% RSLogix 500 project P4_BAK000.RSS, saved by version 8.10.00.18 %
PROJECT "UNTITLED"    % processor: MicroLogix 1200 %

PROGRAM FILES
  LAD 2   4 rungs
  LAD 3 "IO'S"  7 rungs
  LAD 4 "CONTROL"  11 rungs
  LAD 5 "CYCLE'S"  10 rungs

DATA FILES
  O0 OUTPUT  4 elements
  I1 INPUT  4 elements
  S2 STATUS  66 elements
  B3 BINARY  2 elements
  T4 TIMER  3 elements
  C5 COUNTER  1 elements
  R6 CONTROL  1 elements
  N7 INTEGER  2 elements

LADDER 2
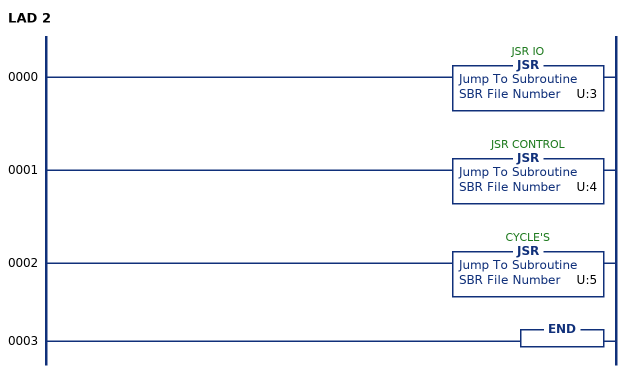
% Rung: 0 %
SOR JSR U:3 EOR
%   U:3  "JSR IO" %
% Rung: 1 %
SOR JSR U:4 EOR
%   U:4  "JSR CONTROL" %
% Rung: 2 %
SOR JSR U:5 EOR
%   U:5  "CYCLE'S" %
% Rung: 3 %
SOR END EOR

LADDER 3 "IO'S"
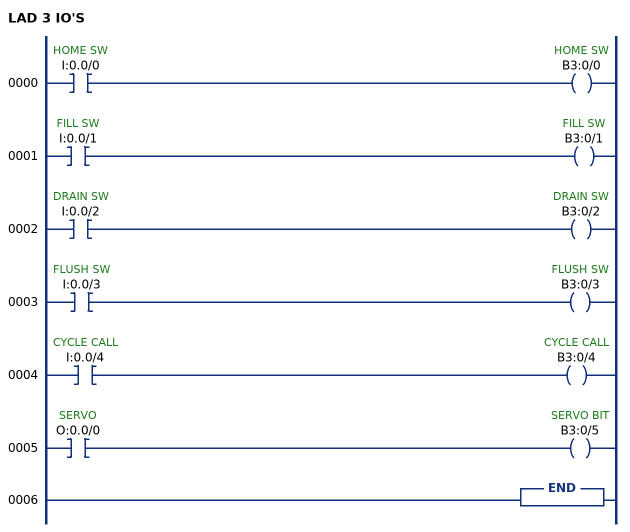
% Rung: 0 %
SOR XIC I:0.0/0 OTE B3:0/0 EOR
%   I:0.0/0  "HOME SW" %
%   B3:0/0  "HOME SW" %
% Rung: 1 %
SOR XIC I:0.0/1 OTE B3:0/1 EOR
%   I:0.0/1  "FILL SW" %
%   B3:0/1  "FILL SW" %
% Rung: 2 %
SOR XIC I:0.0/2 OTE B3:0/2 EOR
%   I:0.0/2  "DRAIN SW" %
%   B3:0/2  "DRAIN SW" %
% Rung: 3 %
SOR XIC I:0.0/3 OTE B3:0/3 EOR
%   I:0.0/3  "FLUSH SW" %
%   B3:0/3  "FLUSH SW" %
% Rung: 4 %
SOR XIC I:0.0/4 OTE B3:0/4 EOR
%   I:0.0/4  "CYCLE CALL" %
%   B3:0/4  "CYCLE CALL" %
% Rung: 5 %
SOR XIC O:0.0/0 OTE B3:0/5 EOR
%   O:0.0/0  "SERVO" %
%   B3:0/5  "SERVO BIT" %
% Rung: 6 %
SOR END EOR

LADDER 4 "CONTROL"
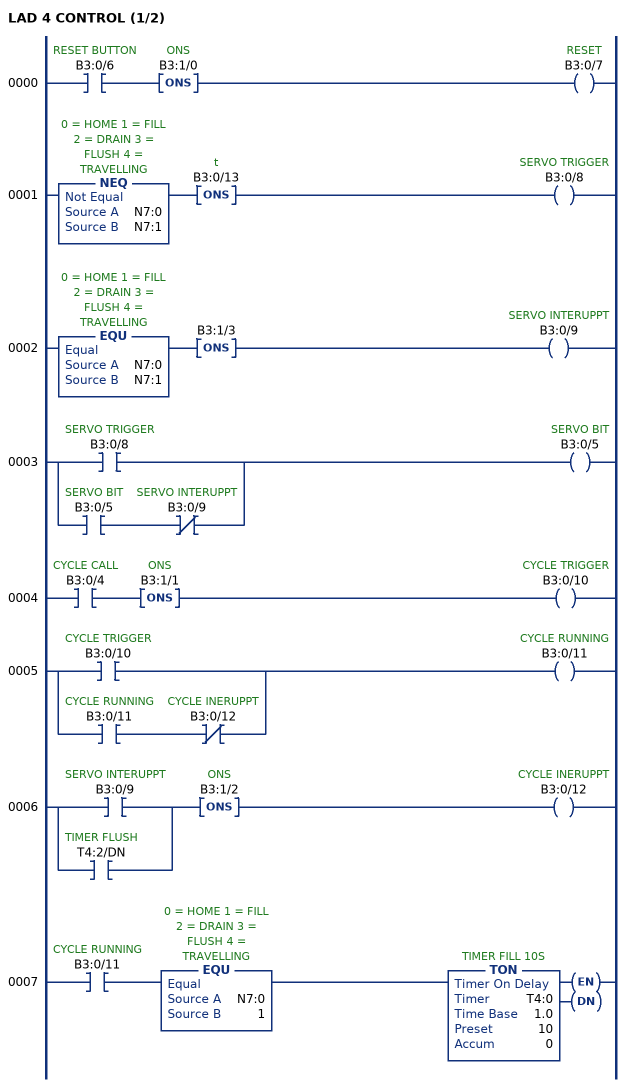
% Rung: 0 %
SOR XIC B3:0/6 ONS B3:1/0 OTE B3:0/7 EOR
%   B3:0/6  "RESET BUTTON" %
%   B3:1/0  "ONS" %
%   B3:0/7  "RESET" %
% Rung: 1 %
SOR NEQ N7:0 N7:1 ONS B3:0/13 OTE B3:0/8 EOR
%   N7:0  "0 = HOME 1 = FILL 2 = DRAIN 3 = FLUSH 4 = TRAVELLING" %
%   N7:1  "DESIRED:    0 = HOME 1 = FILL 2 = DRAIN 3 = FLUSH 4 = TRAVELLING" %
%   B3:0/13  "t" %
%   B3:0/8  "SERVO TRIGGER" %
% Rung: 2 %
SOR EQU N7:0 N7:1 ONS B3:1/3 OTE B3:0/9 EOR
%   N7:0  "0 = HOME 1 = FILL 2 = DRAIN 3 = FLUSH 4 = TRAVELLING" %
%   N7:1  "DESIRED:    0 = HOME 1 = FILL 2 = DRAIN 3 = FLUSH 4 = TRAVELLING" %
%   B3:0/9  "SERVO INTERUPPT" %
% Rung: 3 %
SOR BST XIC B3:0/8 NXB XIC B3:0/5 XIO B3:0/9 BND OTE B3:0/5 EOR
%   B3:0/8  "SERVO TRIGGER" %
%   B3:0/5  "SERVO BIT" %
%   B3:0/9  "SERVO INTERUPPT" %
% Rung: 4 %
SOR XIC B3:0/4 ONS B3:1/1 OTE B3:0/10 EOR
%   B3:0/4  "CYCLE CALL" %
%   B3:1/1  "ONS" %
%   B3:0/10  "CYCLE TRIGGER" %
% Rung: 5 %
SOR BST XIC B3:0/10 NXB XIC B3:0/11 XIO B3:0/12 BND OTE B3:0/11 EOR
%   B3:0/10  "CYCLE TRIGGER" %
%   B3:0/11  "CYCLE RUNNING" %
%   B3:0/12  "CYCLE INERUPPT" %
% Rung: 6 %
SOR BST XIC B3:0/9 NXB XIC T4:2/DN BND ONS B3:1/2 OTE B3:0/12 EOR
%   B3:0/9  "SERVO INTERUPPT" %
%   T4:2  "TIMER FLUSH" %
%   B3:1/2  "ONS" %
%   B3:0/12  "CYCLE INERUPPT" %
% Rung: 7 %
SOR XIC B3:0/11 EQU N7:0 1 TON T4:0 1.0 10 0 EOR
%   B3:0/11  "CYCLE RUNNING" %
%   N7:0  "0 = HOME 1 = FILL 2 = DRAIN 3 = FLUSH 4 = TRAVELLING" %
%   T4:0  "TIMER FILL 10S" %

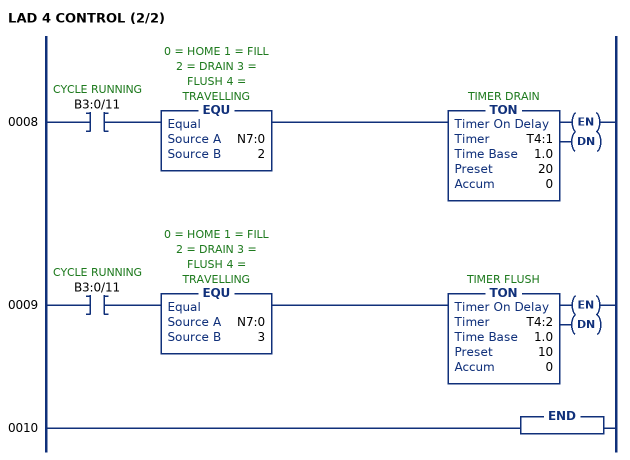
% Rung: 8 %
SOR XIC B3:0/11 EQU N7:0 2 TON T4:1 1.0 20 0 EOR
%   B3:0/11  "CYCLE RUNNING" %
%   N7:0  "0 = HOME 1 = FILL 2 = DRAIN 3 = FLUSH 4 = TRAVELLING" %
%   T4:1  "TIMER DRAIN" %
% Rung: 9 %
SOR XIC B3:0/11 EQU N7:0 3 TON T4:2 1.0 10 0 EOR
%   B3:0/11  "CYCLE RUNNING" %
%   N7:0  "0 = HOME 1 = FILL 2 = DRAIN 3 = FLUSH 4 = TRAVELLING" %
%   T4:2  "TIMER FLUSH" %
% Rung: 10 %
SOR END EOR

LADDER 5 "CYCLE'S"
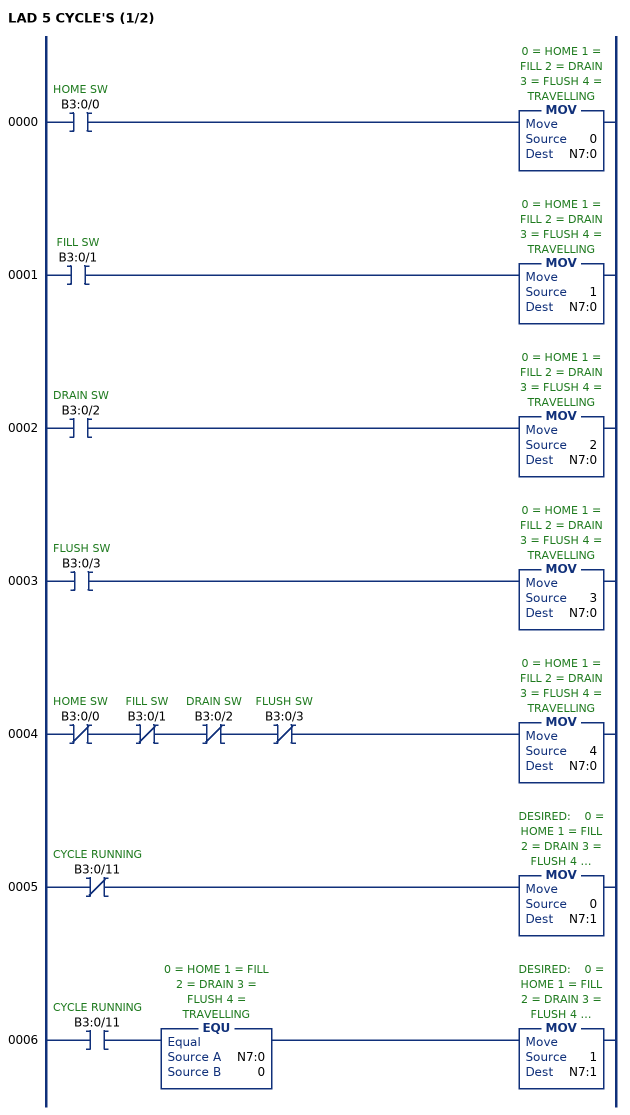
% Rung: 0 %
SOR XIC B3:0/0 MOV 0 N7:0 EOR
%   B3:0/0  "HOME SW" %
%   N7:0  "0 = HOME 1 = FILL 2 = DRAIN 3 = FLUSH 4 = TRAVELLING" %
% Rung: 1 %
SOR XIC B3:0/1 MOV 1 N7:0 EOR
%   B3:0/1  "FILL SW" %
%   N7:0  "0 = HOME 1 = FILL 2 = DRAIN 3 = FLUSH 4 = TRAVELLING" %
% Rung: 2 %
SOR XIC B3:0/2 MOV 2 N7:0 EOR
%   B3:0/2  "DRAIN SW" %
%   N7:0  "0 = HOME 1 = FILL 2 = DRAIN 3 = FLUSH 4 = TRAVELLING" %
% Rung: 3 %
SOR XIC B3:0/3 MOV 3 N7:0 EOR
%   B3:0/3  "FLUSH SW" %
%   N7:0  "0 = HOME 1 = FILL 2 = DRAIN 3 = FLUSH 4 = TRAVELLING" %
% Rung: 4 %
SOR XIO B3:0/0 XIO B3:0/1 XIO B3:0/2 XIO B3:0/3 MOV 4 N7:0 EOR
%   B3:0/0  "HOME SW" %
%   B3:0/1  "FILL SW" %
%   B3:0/2  "DRAIN SW" %
%   B3:0/3  "FLUSH SW" %
%   N7:0  "0 = HOME 1 = FILL 2 = DRAIN 3 = FLUSH 4 = TRAVELLING" %
% Rung: 5 %
SOR XIO B3:0/11 MOV 0 N7:1 EOR
%   B3:0/11  "CYCLE RUNNING" %
%   N7:1  "DESIRED:    0 = HOME 1 = FILL 2 = DRAIN 3 = FLUSH 4 = TRAVELLING" %
% Rung: 6 %
SOR XIC B3:0/11 EQU N7:0 0 MOV 1 N7:1 EOR
%   B3:0/11  "CYCLE RUNNING" %
%   N7:0  "0 = HOME 1 = FILL 2 = DRAIN 3 = FLUSH 4 = TRAVELLING" %
%   N7:1  "DESIRED:    0 = HOME 1 = FILL 2 = DRAIN 3 = FLUSH 4 = TRAVELLING" %

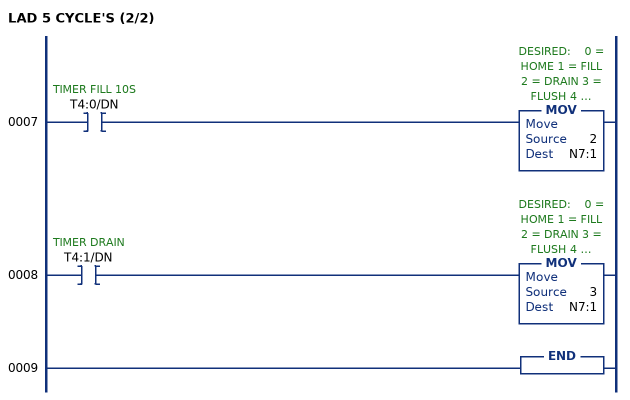
% Rung: 7 %
SOR XIC T4:0/DN MOV 2 N7:1 EOR
%   T4:0  "TIMER FILL 10S" %
%   N7:1  "DESIRED:    0 = HOME 1 = FILL 2 = DRAIN 3 = FLUSH 4 = TRAVELLING" %
% Rung: 8 %
SOR XIC T4:1/DN MOV 3 N7:1 EOR
%   T4:1  "TIMER DRAIN" %
%   N7:1  "DESIRED:    0 = HOME 1 = FILL 2 = DRAIN 3 = FLUSH 4 = TRAVELLING" %
% Rung: 9 %
SOR END EOR

DATA TABLE (non-zero values as saved)
DATA B3
% B3:0 % 0X2002 0X0010
DATA T4
% .PRE .ACC %
% T4:0 % 10 0
% T4:1 % 20 0
% T4:2 % 10 0
DATA N7
% N7:0 % 1 0
